{attribute 'strict'}
TYPE E_AxisStateInit :
(
	AXIS_INIT_RESET		:= 0,	(* Reseting all function blocks *)
	AXIS_INIT_POWER_ON	:= 10,	(* Powering on the axis *)
	AXIS_INIT_DONE		:= 20	(* Initialization done *)
);
END_TYPE

(* stored: Version 1.1.0.1, ProductVersion 3.1.4024.9
   DUT E_AxisStateInit: Id {d5f5a61d-a019-4f4f-917d-6b8a62487a38} *)
